TYPE ST_PNOZCommDiag :
STRUCT
    bitWcState: BIT; //0 = Valid real-time communication in the last cycle, 1 = Invalid real-time communication
    bitInputToggle: BIT; //It changes its state 0/1 whenever new data is received.
    nEtherCATState: UINT; //State of EtherCAT slave
END_STRUCT
END_TYPE

(* stored: Version 1.1.0.1
   DUT ST_PNOZCommDiag: Id {5cc4dacf-5e42-0a6f-2af9-92b983426889} *)
